SYSTEM TRAFFICtester (* System Configuration *)
  (* Standard: 61499-1 *)
  (* Version 0.4, 2009-03-05, JHC, Holobloc Inc., Deleted Application. *)
  (* Version 0.3, 2003-12-05, JHC, Rockwell Automation, Renamed from NEWSYSTEM. *)
  (* Version 0.2, 2002-11-05, JHC, Rockwell Automation, Fixed missing (empty) FBD in Application. *)
  (* Version 0.1, 2002-01-17, JHC, Rockwell Automation, Minor cleanup *)
  (* Version 0.0, 2000-05-27, JHC, Rockwell Automation *)
  DEVICE Device1 : FRAME_DEVICE(BOUNDS := [100,100,300,110])
    RESOURCE HMI : PANEL_RESOURCE
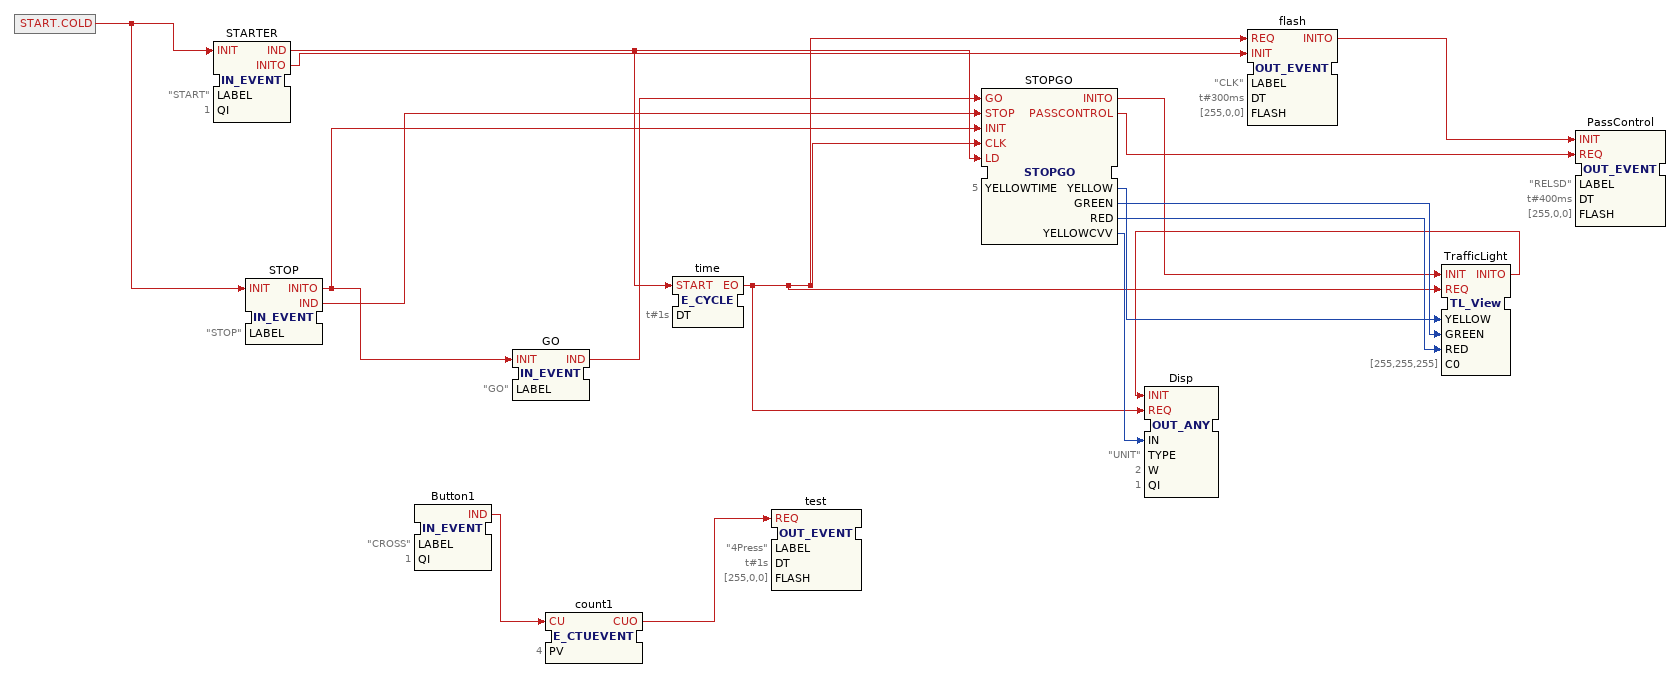
      FBS
        Button1 : IN_EVENT(LABEL := "CROSS", QI := 1);
        count1 : E_CTUEVENT(PV := 4);
        test : OUT_EVENT(LABEL := "4Press", DT := t#1s, FLASH := [255,0,0]);
        TrafficLight : TL_View(C0 := [255,255,255]);
        STOPGO : STOPGO(YELLOWTIME := 5);
        STOP : IN_EVENT(LABEL := "STOP");
        GO : IN_EVENT(LABEL := "GO");
        time : E_CYCLE(DT := t#1s);
        STARTER : IN_EVENT(LABEL := "START", QI := 1);
        flash : OUT_EVENT(LABEL := "CLK", DT := t#300ms, FLASH := [255,0,0]);
        Disp : OUT_ANY(TYPE := "UNIT", W := 2, QI := 1);
        PassControl : OUT_EVENT(LABEL := "RELSD", DT := t#400ms, FLASH := [255,0,0]);
      END_FBS
      EVENT_CONNECTIONS
        Button1.IND TO count1.CU;
        count1.CUO TO test.REQ;
        STOPGO.INITO TO TrafficLight.INIT;
        START.COLD TO STOP.INIT;
        STOP.INITO TO GO.INIT;
        GO.IND TO STOPGO.GO;
        STOP.IND TO STOPGO.STOP;
        STOP.INITO TO STOPGO.INIT;
        time.EO TO STOPGO.CLK;
        START.COLD TO STARTER.INIT;
        STARTER.IND TO time.START;
        time.EO TO flash.REQ;
        STARTER.INITO TO flash.INIT;
        time.EO TO TrafficLight.REQ;
        TrafficLight.INITO TO Disp.INIT;
        time.EO TO Disp.REQ;
        STARTER.IND TO STOPGO.LD;
        flash.INITO TO PassControl.INIT;
        STOPGO.PASSCONTROL TO PassControl.REQ;
      END_CONNECTIONS
      DATA_CONNECTIONS
        STOPGO.YELLOW TO TrafficLight.YELLOW;
        STOPGO.GREEN TO TrafficLight.GREEN;
        STOPGO.RED TO TrafficLight.RED;
        STOPGO.YELLOWCVV TO Disp.IN;
      END_CONNECTIONS
    END_RESOURCE
  END_DEVICE
END_SYSTEM
